{attribute addProperty BoxType "EL2521--0000"}
{attribute addProperty Id "InputsAT %I*Inputs_406D1DC23240OutputsAT %Q*Outputs_5374A1F83240WcStateAT %I*WcState_F855686C1620InfoDataAT %I*InfoData_BC63D37F80100"}
{attribute addProperty CRC "3548921766"}
{attribute addProperty SizeInBites "160"}
{attribute addProperty SizeInBytes "20"}
TYPE EL2521_1302708C :
STRUCT
	{attribute addProperty Name "Inputs"}
	Inputs : Inputs_406D1DC2;
	{attribute addProperty Name "Outputs"}
	Outputs : Outputs_5374A1F8;
	{attribute addProperty Name "WcState"}
	WcState : WcState_F855686C;
	{attribute addProperty Name "InfoData"}
	InfoData : InfoData_BC63D37F;
END_STRUCT
END_TYPE

(* stored: Version 1.2.0.0, ProductVersion 3.1.4024.9
   DUT EL2521_1302708C: Id {74aa13ce-9854-4ef8-b6a7-5f6322450162} *)
